{attribute 'qualified_only'}
VAR_GLOBAL
	// set level to log. Lower log level includes higher levels i.e. info does warning and Error. 
	LogLevel : E_LogSeverity_Ish := E_LogSeverity_Ish.Error; // Turn messages off by default

END_VAR

(* stored: Version 1.1.0.1, ProductVersion 3.1.4022.18
   GVL LogConfig: Id {7c65e267-1db9-41c8-90bc-d0c05ea63b98} *)
